// TIA Portal V18 export
// export: Created 2026-06-07T17:03:10.0178191Z, ExportSetting WithDefaults, DisplayName Totally Integrated Automation Portal, DisplayVersion V18, DisplayName TIA Portal Openness, DisplayVersion V18, DisplayName TIA Portal Version Control Interface, DisplayVersion V18, DisplayName STEP 7 Professional, DisplayVersion V18, DisplayName STEP 7 Safety, DisplayVersion V18, DisplayName WinCC Professional, DisplayVersion V18
ORGANIZATION_BLOCK "Main"   // OB1, LAD, ProgramCycle
TITLE = "Main Program Sweep (Cycle)"
{ S7_Optimized_Access := 'TRUE' }
VERSION : 0.1
// stored: AutoNumber true, IsIECCheckEnabled false, SetENOAutomatically false
   VAR_INPUT
      Initial_Call : Bool;   // Initial call of this OB
      Remanence : Bool;   // =True, if remanent data are available
   END_VAR
BEGIN

REGION Network 1
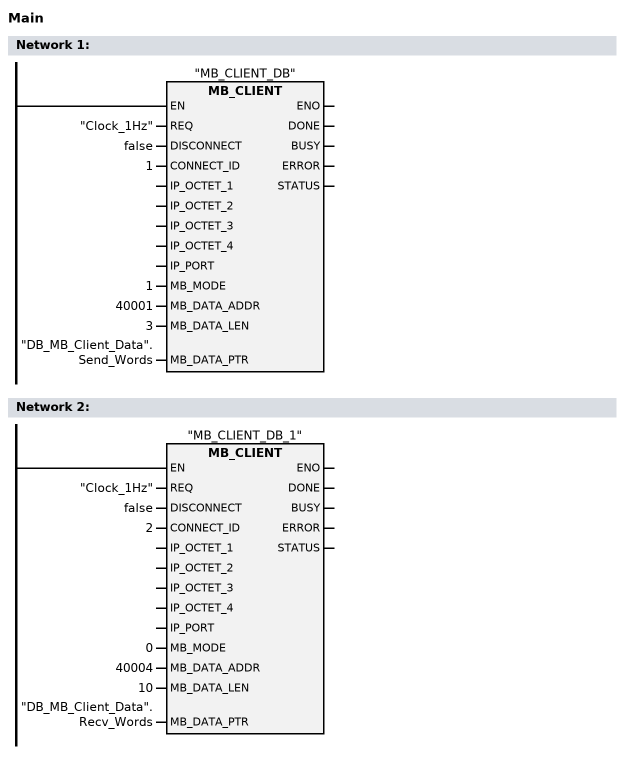
   RUNG wire#powerrail
      { S7_Templates := "[card1200 := 1, card1500 := 0]" } "MB_CLIENT_DB".MB_CLIENT(REQ := "Clock_1Hz", DISCONNECT := false, CONNECT_ID := 1, IP_OCTET_1 :=, IP_OCTET_2 :=, IP_OCTET_3 :=, IP_OCTET_4 :=, IP_PORT :=, MB_MODE := 1, MB_DATA_ADDR := 40001, MB_DATA_LEN := 3, MB_DATA_PTR := "DB_MB_Client_Data".Send_Words, DONE =>, BUSY =>, ERROR =>, STATUS =>)
   END_RUNG
   // the same network as SCL:
   "MB_CLIENT_DB"(REQ := "Clock_1Hz",   // MB_CLIENT
                  DISCONNECT := false,
                  CONNECT_ID := 1,
                  MB_MODE := 1,
                  MB_DATA_ADDR := 40001,
                  MB_DATA_LEN := 3,
                  MB_DATA_PTR := "DB_MB_Client_Data".Send_Words);
END_REGION

REGION Network 2
   RUNG wire#powerrail
      { S7_Templates := "[card1200 := 1, card1500 := 0]" } "MB_CLIENT_DB_1".MB_CLIENT(REQ := "Clock_1Hz", DISCONNECT := false, CONNECT_ID := 2, IP_OCTET_1 :=, IP_OCTET_2 :=, IP_OCTET_3 :=, IP_OCTET_4 :=, IP_PORT :=, MB_MODE := 0, MB_DATA_ADDR := 40004, MB_DATA_LEN := 10, MB_DATA_PTR := "DB_MB_Client_Data".Recv_Words, DONE =>, BUSY =>, ERROR =>, STATUS =>)
   END_RUNG
   // the same network as SCL:
   "MB_CLIENT_DB_1"(REQ := "Clock_1Hz",   // MB_CLIENT
                    DISCONNECT := false,
                    CONNECT_ID := 2,
                    MB_MODE := 0,
                    MB_DATA_ADDR := 40004,
                    MB_DATA_LEN := 10,
                    MB_DATA_PTR := "DB_MB_Client_Data".Recv_Words);
END_REGION
END_ORGANIZATION_BLOCK
